// TIA Portal V17 export
// export: Created 2023-12-29T10:44:22.8737876Z, ExportSetting None, DisplayName Totally Integrated Automation Portal, DisplayVersion V17 Update 4, DisplayName TIA Portal Openness, DisplayVersion V17 Update 4, DisplayName TIA Portal Version Control Interface, DisplayVersion V17, DisplayName STEP 7 Professional, DisplayVersion V17 Update 4, DisplayName STEP 7 Safety, DisplayVersion V17, DisplayName WinCC Advanced / Unified PC, DisplayVersion V17 Update 4
FUNCTION "FC_AIn2oo3" : Void   // FC31, LAD
{ S7_Optimized_Access := 'FALSE' }
// AnalogInput2oo3
// stored: AutoNumber false, SetENOAutomatically false
BEGIN

REGION Network 1: AI 1
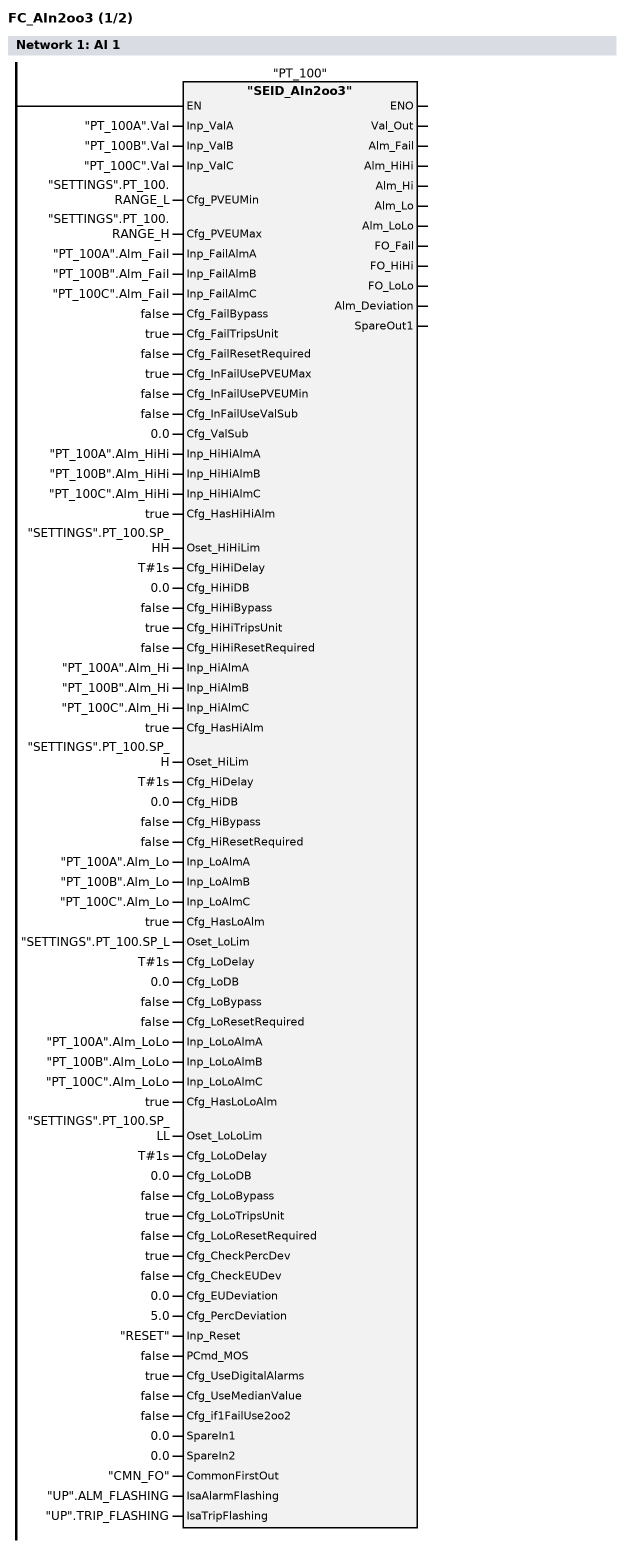
   RUNG wire#powerrail
      "PT_100"(Inp_ValA := "PT_100A".Val, Inp_ValB := "PT_100B".Val, Inp_ValC := "PT_100C".Val, Cfg_PVEUMin := "SETTINGS".PT_100.RANGE_L, Cfg_PVEUMax := "SETTINGS".PT_100.RANGE_H, Inp_FailAlmA := "PT_100A".Alm_Fail, Inp_FailAlmB := "PT_100B".Alm_Fail, Inp_FailAlmC := "PT_100C".Alm_Fail, Cfg_FailBypass := false, Cfg_FailTripsUnit := true, Cfg_FailResetRequired := false, Cfg_InFailUsePVEUMax := true, Cfg_InFailUsePVEUMin := false, Cfg_InFailUseValSub := false, Cfg_ValSub := 0.0, Inp_HiHiAlmA := "PT_100A".Alm_HiHi, Inp_HiHiAlmB := "PT_100B".Alm_HiHi, Inp_HiHiAlmC := "PT_100C".Alm_HiHi, Cfg_HasHiHiAlm := true, Oset_HiHiLim := "SETTINGS".PT_100.SP_HH, Cfg_HiHiDelay := T#1s, Cfg_HiHiDB := 0.0, Cfg_HiHiBypass := false, Cfg_HiHiTripsUnit := true, Cfg_HiHiResetRequired := false, Inp_HiAlmA := "PT_100A".Alm_Hi, Inp_HiAlmB := "PT_100B".Alm_Hi, Inp_HiAlmC := "PT_100C".Alm_Hi, Cfg_HasHiAlm := true, Oset_HiLim := "SETTINGS".PT_100.SP_H, Cfg_HiDelay := T#1s, Cfg_HiDB := 0.0, Cfg_HiBypass := false, Cfg_HiResetRequired := false, Inp_LoAlmA := "PT_100A".Alm_Lo, Inp_LoAlmB := "PT_100B".Alm_Lo, Inp_LoAlmC := "PT_100C".Alm_Lo, Cfg_HasLoAlm := true, Oset_LoLim := "SETTINGS".PT_100.SP_L, Cfg_LoDelay := T#1s, Cfg_LoDB := 0.0, Cfg_LoBypass := false, Cfg_LoResetRequired := false, Inp_LoLoAlmA := "PT_100A".Alm_LoLo, Inp_LoLoAlmB := "PT_100B".Alm_LoLo, Inp_LoLoAlmC := "PT_100C".Alm_LoLo, Cfg_HasLoLoAlm := true, Oset_LoLoLim := "SETTINGS".PT_100.SP_LL, Cfg_LoLoDelay := T#1s, Cfg_LoLoDB := 0.0, Cfg_LoLoBypass := false, Cfg_LoLoTripsUnit := true, Cfg_LoLoResetRequired := false, Cfg_CheckPercDev := true, Cfg_CheckEUDev := false, Cfg_EUDeviation := 0.0, Cfg_PercDeviation := 5.0, Inp_Reset := "RESET", PCmd_MOS := false, Cfg_UseDigitalAlarms := true, Cfg_UseMedianValue := false, Cfg_if1FailUse2oo2 := false, SpareIn1 := 0.0, SpareIn2 := 0.0, CommonFirstOut := "CMN_FO", IsaAlarmFlashing := "UP".ALM_FLASHING, IsaTripFlashing := "UP".TRIP_FLASHING, Val_Out =>, Alm_Fail =>, Alm_HiHi =>, Alm_Hi =>, Alm_Lo =>, Alm_LoLo =>, FO_Fail =>, FO_HiHi =>, FO_LoLo =>, Alm_Deviation =>, SpareOut1 =>)
   END_RUNG
   // the same network as SCL:
   "PT_100"(Inp_ValA := "PT_100A".Val,   // "SEID_AIn2oo3"
            Inp_ValB := "PT_100B".Val,
            Inp_ValC := "PT_100C".Val,
            Cfg_PVEUMin := "SETTINGS".PT_100.RANGE_L,
            Cfg_PVEUMax := "SETTINGS".PT_100.RANGE_H,
            Inp_FailAlmA := "PT_100A".Alm_Fail,
            Inp_FailAlmB := "PT_100B".Alm_Fail,
            Inp_FailAlmC := "PT_100C".Alm_Fail,
            Cfg_FailBypass := false,
            Cfg_FailTripsUnit := true,
            Cfg_FailResetRequired := false,
            Cfg_InFailUsePVEUMax := true,
            Cfg_InFailUsePVEUMin := false,
            Cfg_InFailUseValSub := false,
            Cfg_ValSub := 0.0,
            Inp_HiHiAlmA := "PT_100A".Alm_HiHi,
            Inp_HiHiAlmB := "PT_100B".Alm_HiHi,
            Inp_HiHiAlmC := "PT_100C".Alm_HiHi,
            Cfg_HasHiHiAlm := true,
            Oset_HiHiLim := "SETTINGS".PT_100.SP_HH,
            Cfg_HiHiDelay := T#1s,
            Cfg_HiHiDB := 0.0,
            Cfg_HiHiBypass := false,
            Cfg_HiHiTripsUnit := true,
            Cfg_HiHiResetRequired := false,
            Inp_HiAlmA := "PT_100A".Alm_Hi,
            Inp_HiAlmB := "PT_100B".Alm_Hi,
            Inp_HiAlmC := "PT_100C".Alm_Hi,
            Cfg_HasHiAlm := true,
            Oset_HiLim := "SETTINGS".PT_100.SP_H,
            Cfg_HiDelay := T#1s,
            Cfg_HiDB := 0.0,
            Cfg_HiBypass := false,
            Cfg_HiResetRequired := false,
            Inp_LoAlmA := "PT_100A".Alm_Lo,
            Inp_LoAlmB := "PT_100B".Alm_Lo,
            Inp_LoAlmC := "PT_100C".Alm_Lo,
            Cfg_HasLoAlm := true,
            Oset_LoLim := "SETTINGS".PT_100.SP_L,
            Cfg_LoDelay := T#1s,
            Cfg_LoDB := 0.0,
            Cfg_LoBypass := false,
            Cfg_LoResetRequired := false,
            Inp_LoLoAlmA := "PT_100A".Alm_LoLo,
            Inp_LoLoAlmB := "PT_100B".Alm_LoLo,
            Inp_LoLoAlmC := "PT_100C".Alm_LoLo,
            Cfg_HasLoLoAlm := true,
            Oset_LoLoLim := "SETTINGS".PT_100.SP_LL,
            Cfg_LoLoDelay := T#1s,
            Cfg_LoLoDB := 0.0,
            Cfg_LoLoBypass := false,
            Cfg_LoLoTripsUnit := true,
            Cfg_LoLoResetRequired := false,
            Cfg_CheckPercDev := true,
            Cfg_CheckEUDev := false,
            Cfg_EUDeviation := 0.0,
            Cfg_PercDeviation := 5.0,
            Inp_Reset := "RESET",
            PCmd_MOS := false,
            Cfg_UseDigitalAlarms := true,
            Cfg_UseMedianValue := false,
            Cfg_if1FailUse2oo2 := false,
            SpareIn1 := 0.0,
            SpareIn2 := 0.0,
            CommonFirstOut := "CMN_FO",
            IsaAlarmFlashing := "UP".ALM_FLASHING,
            IsaTripFlashing := "UP".TRIP_FLASHING);
END_REGION

REGION Network 2: AI 3
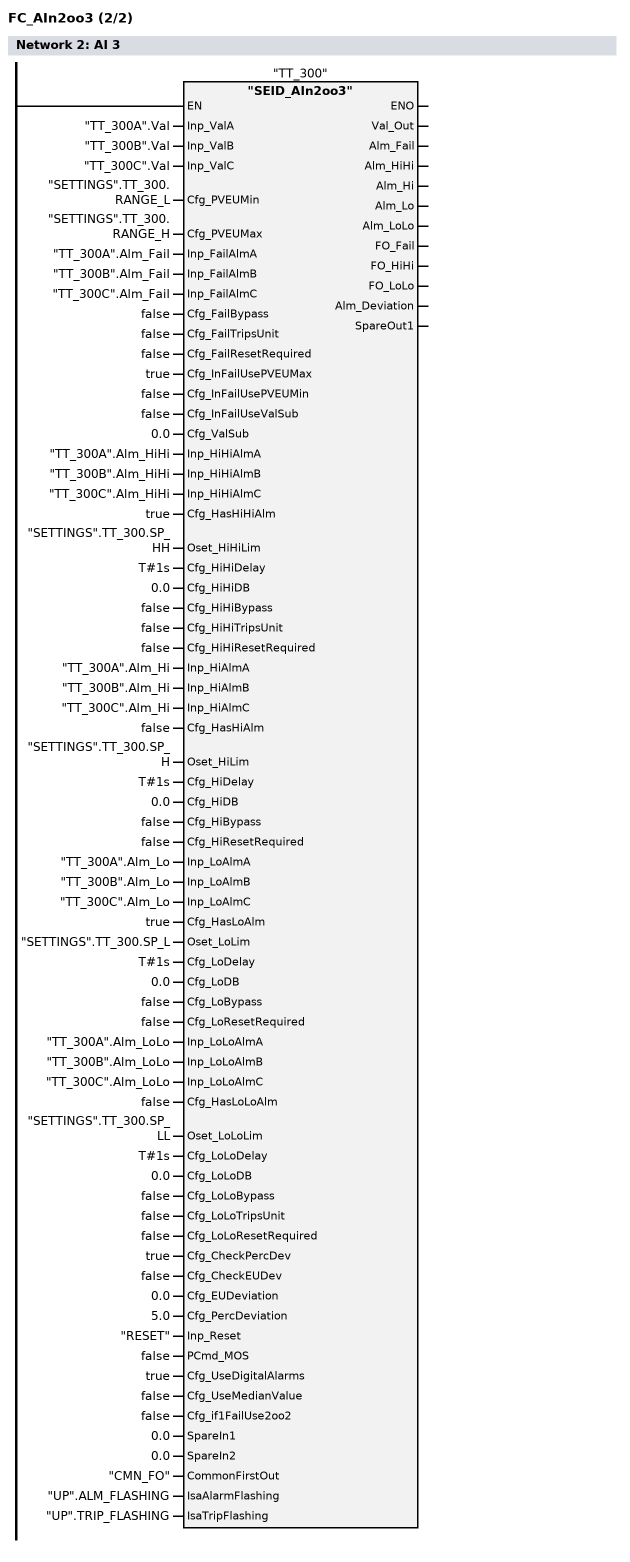
   RUNG wire#powerrail
      "TT_300"(Inp_ValA := "TT_300A".Val, Inp_ValB := "TT_300B".Val, Inp_ValC := "TT_300C".Val, Cfg_PVEUMin := "SETTINGS".TT_300.RANGE_L, Cfg_PVEUMax := "SETTINGS".TT_300.RANGE_H, Inp_FailAlmA := "TT_300A".Alm_Fail, Inp_FailAlmB := "TT_300B".Alm_Fail, Inp_FailAlmC := "TT_300C".Alm_Fail, Cfg_FailBypass := false, Cfg_FailTripsUnit := false, Cfg_FailResetRequired := false, Cfg_InFailUsePVEUMax := true, Cfg_InFailUsePVEUMin := false, Cfg_InFailUseValSub := false, Cfg_ValSub := 0.0, Inp_HiHiAlmA := "TT_300A".Alm_HiHi, Inp_HiHiAlmB := "TT_300B".Alm_HiHi, Inp_HiHiAlmC := "TT_300C".Alm_HiHi, Cfg_HasHiHiAlm := true, Oset_HiHiLim := "SETTINGS".TT_300.SP_HH, Cfg_HiHiDelay := T#1s, Cfg_HiHiDB := 0.0, Cfg_HiHiBypass := false, Cfg_HiHiTripsUnit := false, Cfg_HiHiResetRequired := false, Inp_HiAlmA := "TT_300A".Alm_Hi, Inp_HiAlmB := "TT_300B".Alm_Hi, Inp_HiAlmC := "TT_300C".Alm_Hi, Cfg_HasHiAlm := false, Oset_HiLim := "SETTINGS".TT_300.SP_H, Cfg_HiDelay := T#1s, Cfg_HiDB := 0.0, Cfg_HiBypass := false, Cfg_HiResetRequired := false, Inp_LoAlmA := "TT_300A".Alm_Lo, Inp_LoAlmB := "TT_300B".Alm_Lo, Inp_LoAlmC := "TT_300C".Alm_Lo, Cfg_HasLoAlm := true, Oset_LoLim := "SETTINGS".TT_300.SP_L, Cfg_LoDelay := T#1s, Cfg_LoDB := 0.0, Cfg_LoBypass := false, Cfg_LoResetRequired := false, Inp_LoLoAlmA := "TT_300A".Alm_LoLo, Inp_LoLoAlmB := "TT_300B".Alm_LoLo, Inp_LoLoAlmC := "TT_300C".Alm_LoLo, Cfg_HasLoLoAlm := false, Oset_LoLoLim := "SETTINGS".TT_300.SP_LL, Cfg_LoLoDelay := T#1s, Cfg_LoLoDB := 0.0, Cfg_LoLoBypass := false, Cfg_LoLoTripsUnit := false, Cfg_LoLoResetRequired := false, Cfg_CheckPercDev := true, Cfg_CheckEUDev := false, Cfg_EUDeviation := 0.0, Cfg_PercDeviation := 5.0, Inp_Reset := "RESET", PCmd_MOS := false, Cfg_UseDigitalAlarms := true, Cfg_UseMedianValue := false, Cfg_if1FailUse2oo2 := false, SpareIn1 := 0.0, SpareIn2 := 0.0, CommonFirstOut := "CMN_FO", IsaAlarmFlashing := "UP".ALM_FLASHING, IsaTripFlashing := "UP".TRIP_FLASHING, Val_Out =>, Alm_Fail =>, Alm_HiHi =>, Alm_Hi =>, Alm_Lo =>, Alm_LoLo =>, FO_Fail =>, FO_HiHi =>, FO_LoLo =>, Alm_Deviation =>, SpareOut1 =>)
   END_RUNG
   // the same network as SCL:
   "TT_300"(Inp_ValA := "TT_300A".Val,   // "SEID_AIn2oo3"
            Inp_ValB := "TT_300B".Val,
            Inp_ValC := "TT_300C".Val,
            Cfg_PVEUMin := "SETTINGS".TT_300.RANGE_L,
            Cfg_PVEUMax := "SETTINGS".TT_300.RANGE_H,
            Inp_FailAlmA := "TT_300A".Alm_Fail,
            Inp_FailAlmB := "TT_300B".Alm_Fail,
            Inp_FailAlmC := "TT_300C".Alm_Fail,
            Cfg_FailBypass := false,
            Cfg_FailTripsUnit := false,
            Cfg_FailResetRequired := false,
            Cfg_InFailUsePVEUMax := true,
            Cfg_InFailUsePVEUMin := false,
            Cfg_InFailUseValSub := false,
            Cfg_ValSub := 0.0,
            Inp_HiHiAlmA := "TT_300A".Alm_HiHi,
            Inp_HiHiAlmB := "TT_300B".Alm_HiHi,
            Inp_HiHiAlmC := "TT_300C".Alm_HiHi,
            Cfg_HasHiHiAlm := true,
            Oset_HiHiLim := "SETTINGS".TT_300.SP_HH,
            Cfg_HiHiDelay := T#1s,
            Cfg_HiHiDB := 0.0,
            Cfg_HiHiBypass := false,
            Cfg_HiHiTripsUnit := false,
            Cfg_HiHiResetRequired := false,
            Inp_HiAlmA := "TT_300A".Alm_Hi,
            Inp_HiAlmB := "TT_300B".Alm_Hi,
            Inp_HiAlmC := "TT_300C".Alm_Hi,
            Cfg_HasHiAlm := false,
            Oset_HiLim := "SETTINGS".TT_300.SP_H,
            Cfg_HiDelay := T#1s,
            Cfg_HiDB := 0.0,
            Cfg_HiBypass := false,
            Cfg_HiResetRequired := false,
            Inp_LoAlmA := "TT_300A".Alm_Lo,
            Inp_LoAlmB := "TT_300B".Alm_Lo,
            Inp_LoAlmC := "TT_300C".Alm_Lo,
            Cfg_HasLoAlm := true,
            Oset_LoLim := "SETTINGS".TT_300.SP_L,
            Cfg_LoDelay := T#1s,
            Cfg_LoDB := 0.0,
            Cfg_LoBypass := false,
            Cfg_LoResetRequired := false,
            Inp_LoLoAlmA := "TT_300A".Alm_LoLo,
            Inp_LoLoAlmB := "TT_300B".Alm_LoLo,
            Inp_LoLoAlmC := "TT_300C".Alm_LoLo,
            Cfg_HasLoLoAlm := false,
            Oset_LoLoLim := "SETTINGS".TT_300.SP_LL,
            Cfg_LoLoDelay := T#1s,
            Cfg_LoLoDB := 0.0,
            Cfg_LoLoBypass := false,
            Cfg_LoLoTripsUnit := false,
            Cfg_LoLoResetRequired := false,
            Cfg_CheckPercDev := true,
            Cfg_CheckEUDev := false,
            Cfg_EUDeviation := 0.0,
            Cfg_PercDeviation := 5.0,
            Inp_Reset := "RESET",
            PCmd_MOS := false,
            Cfg_UseDigitalAlarms := true,
            Cfg_UseMedianValue := false,
            Cfg_if1FailUse2oo2 := false,
            SpareIn1 := 0.0,
            SpareIn2 := 0.0,
            CommonFirstOut := "CMN_FO",
            IsaAlarmFlashing := "UP".ALM_FLASHING,
            IsaTripFlashing := "UP".TRIP_FLASHING);
END_REGION
END_FUNCTION
